DATA_BLOCK "FB_HVAC_Runtime_DB"
{ S7_Optimized_Access := 'FALSE' }
VERSION : 1.0
NON_RETAIN
"FB_HVAC_Runtime"

BEGIN

END_DATA_BLOCK
